# EPICS autosave request: tests/testfiles/cfg/SF_UIND_PV.req
$(SYS):K_SET
$(SYS):GAP_SP
$(SYS):GM-X-SET
$(SYS):GM-Y-SET
$(SYS):GM-PITCH-SET
$(SYS):GM-YAW-SET
$(SYS):GM-ROLL-SET
$(SYS):I-SET
$(SYS):PHI_SET
